# EPICS autosave request: ADApp/Db/pvaDriver_settings.req
$(P)$(R)PvName
file "ADBase_settings.req", P=$(P), R=$(R)
